FUNCTION_BLOCK FB_AND (* Boolean AND *)
  (* Standard: 61499-1-D.1; Classification: Boolean functions *)
  (* Version 0.1, 2001-08-05, JHC, Rockwell Automation, XML version *)
  (* Version 0.0, 1999-02-20, JHC, Rockwell Automation, SRC version *)
  (* Compiler header: package fb.rt.math; *)
  (* Compiler classdef: class FB_AND extends FBFunction2 *)
  (* Compiler Java IBM VisualAge 3.0 *)
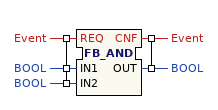
  EVENT_INPUT
    REQ WITH IN1, IN2;
  END_EVENT
  EVENT_OUTPUT
    CNF WITH OUT;
  END_EVENT
  VAR_INPUT
    IN1 : BOOL;
    IN2 : BOOL;
  END_VAR
  VAR_OUTPUT
    OUT : BOOL; (* Result *)
  END_VAR
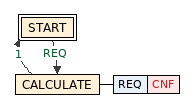
  EC_STATES
    START;
    CALCULATE : REQ -> CNF;
  END_STATES
  EC_TRANSITIONS
    START TO CALCULATE := REQ;
    CALCULATE TO START := 1;
  END_TRANSITIONS
  ALGORITHM REQ IN JAVA:
OUT.setValue(IN1.getValue()&IN2.getValue());
  END_ALGORITHM
END_FUNCTION_BLOCK
